ABB RobotStudio station: HackZurich_20170915-223747.rsstn

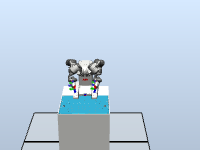
Station HackZurich (saved by RobotStudio 6.5.7530.2005)
Controller IRB_14000_0.5kg_0.5m_1, task T_ROB_L: task frame (RAPID world) sits at (0, 0, 832) mm in the station
Controller IRB_14000_0.5kg_0.5m_1, task T_ROB_R: task frame (RAPID world) sits at (0, 0, 832) mm in the station
Controller IRB_14000_0.5kg_0.5m_1
  mechanical unit ROB_R: IRB14000_0.5_0.5_R, 6 joints, base frame (0, 0, 0) mm
  mechanical unit ROB_R_7: IRB14000_0.5_0.5_R, 1 joints, base frame (0, 0, 0) mm
  mechanical unit ROB_L: IRB14000_0.5_0.5_L, 6 joints, base frame (0, 0, 0) mm
  mechanical unit ROB_L_7: IRB14000_0.5_0.5_L, 1 joints, base frame (0, 0, 0) mm
Layout (positions relative to the parent item):
  - SmartGripper_YuM_R [smart component] at (-9.58, -182.61, 1030.63) mm, rotated rx 179.34 ry -63.63 rz 15.45 deg
      signals: DI di_GripperClose, DI di_GripperOpen, GO SG_hand_ActualPosition, GO SG_hand_SysState, DO SG_hand_StatusCalibrated, GO SG_hand_SoftwareVersion, GO SG_hand_ActualSpeed, GI SG_hand_CmdGripper, GI SG_hand_MaxPosition, GI SG_hand_MinPosition
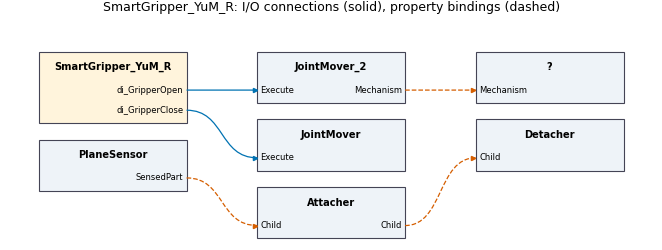
      connections:
        SmartGripper_YuM_R.di_GripperOpen -> JointMover_2.Execute
        SmartGripper_YuM_R.di_GripperClose -> JointMover.Execute
        PlaneSensor.SensedPart => Attacher.Child
        Attacher.Child => Detacher.Child
        JointMover_2.Mechanism => ?.Mechanism
    - PlaneSensor [smart component, from Components\PlaneSensor.rslib]
        properties: Origin=[-0.01 0 0.1]; Axis1=[0 0 0.03]; Axis2=[0.02 0 0]; SensedPart=DownFinger
      - _sensorPart_ [part]
    - Attacher [smart component, from Components\Attacher.rslib]
        properties: Parent=(none); Flange=0; Child=DownFinger; Mount=false; Offset=[0 0 0]; Orientation=[0 0 0]
    - Detacher [smart component, from Components\Detacher.rslib]
        properties: Child=DownFinger; KeepPosition=true
    - JointMover [smart component, from Components\JointMover.rslib]
        properties: Mechanism=YuMi_Hand_R; Relative=false; Duration=1; J1=0
    - JointMover_2 [smart component, from Components\JointMover.rslib]
        properties: Mechanism=YuMi_Hand_R; Relative=false; Duration=1; J1=0.025
    - YuMi_Hand_R [mechanism] at (0, 0, 0) mm; joint values [0] (rad or m)
        TCP Servo at (0, 0, 114.2) mm
        TCP VaccumOne at (56, 18.5, 37.5) mm, rotated rx 0 ry 90 rz 0 deg
        TCP Camera at (-7.3, 28.3, 35.1) mm, rotated rx 0 ry 90 rz 90 deg
        links: HandBase, DownFinger, UpFinger
  - SmartGripper_YuMi_L [smart component] at (-9.58, 182.61, 1030.63) mm, rotated rx -179.34 ry -63.63 rz -15.45 deg
      signals: DI di_GripperClose, DI di_GripperOpen, GO SG_hand_ActualPosition, GO SG_hand_SysState, DO SG_hand_StatusCalibrated, GO SG_hand_SoftwareVersion, GO SG_hand_ActualSpeed, GI SG_hand_CmdGripper, GI SG_hand_MaxPosition, GI SG_hand_MinPosition
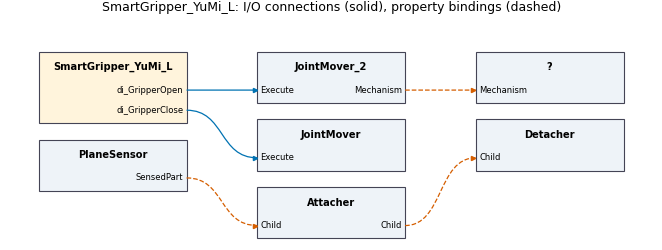
      connections:
        SmartGripper_YuMi_L.di_GripperOpen -> JointMover_2.Execute
        SmartGripper_YuMi_L.di_GripperClose -> JointMover.Execute
        PlaneSensor.SensedPart => Attacher.Child
        Attacher.Child => Detacher.Child
        JointMover_2.Mechanism => ?.Mechanism
    - PlaneSensor [smart component, from Components\PlaneSensor.rslib]
        properties: Origin=[-0.01 0 0.1]; Axis1=[0 0 0.03]; Axis2=[0.02 0 0]; SensedPart=DownFinger
      - _sensorPart_ [part]
    - Attacher [smart component, from Components\Attacher.rslib]
        properties: Parent=(none); Flange=0; Child=DownFinger; Mount=false; Offset=[0 0 0]; Orientation=[0 0 0]
    - Detacher [smart component, from Components\Detacher.rslib]
        properties: Child=DownFinger; KeepPosition=true
    - JointMover [smart component, from Components\JointMover.rslib]
        properties: Mechanism=YuMi_Hand_R; Relative=false; Duration=1; J1=0
    - JointMover_2 [smart component, from Components\JointMover.rslib]
        properties: Mechanism=YuMi_Hand_R; Relative=false; Duration=1; J1=0.025
    - YuMi_Hand_R [mechanism] at (0, 0, 0) mm; joint values [0] (rad or m)
        TCP Servo at (0, 0, 114.2) mm
        TCP VaccumOne at (56, 18.5, 37.5) mm, rotated rx 0 ry 90 rz 0 deg
        TCP Camera at (-7.3, 28.3, 35.1) mm, rotated rx 0 ry 90 rz 90 deg
        links: HandBase, DownFinger, UpFinger
  - IRB14000_0.5_0.5 [mechanism, from Robots\IRB14000_0.5_0.5__01.rslib] at (0, 0, 832) mm
  - IRB14000_0.5_0.5_R [mechanism, from Robots\IRB14000_0.5_0.5__01.rslib] at (0, 0, 832) mm; joint values [0, -2.2689, -2.3562, 0.5236, 0, 0.6981, 0] (rad or m)
  - IRB14000_0.5_0.5_L [mechanism, from Robots\IRB14000_0.5_0.5__01.rslib] at (0, 0, 832) mm; joint values [0, -2.2689, 2.3562, 0.5236, 0, 0.6981, 0] (rad or m)
  - 3HDA000058A6697 | YuMi-Tisch |   Lead Through mit Heberollen [graphiccomponentgroup] at (563, -309.12, 0) mm, rotated rx 0 ry 0 rz 94.33 deg
    - 3HDA000058A6699 | Rahmengestell |   YuMi:1 [graphiccomponentgroup]
      - 3HDA000058A4123 | ITEM Profil8 40x40 |  PROFIL 8 40X40 LEICHT, NATUR:1 [part] at (577.2, -60.29, 36) mm, rotated rx 0 ry -90 rz -3.99 deg
      - 3HDA000058A4123 | ITEM Profil8 40x40 |  PROFIL 8 40X40 LEICHT, NATUR:2 [part] at (577.2, -60.29, 796) mm, rotated rx 0 ry -90 rz -3.99 deg
      - 3HDA000057A1904 |Winkelsatz 8 |  WINKELSATZ 8 80X80 80x80:32 [part] at (621.28, -3.21, 736) mm, rotated rx 180 ry 0 rz 86.01 deg
      - 3HDA000057A1904 |Winkelsatz 8 |  WINKELSATZ 8 80X80 80x80:33 [part] at (716.12, 782.09, 736) mm, rotated rx 180 ry 0 rz -93.99 deg
      - 3HDA000057A1904 |Winkelsatz 8 |  WINKELSATZ 8 80X80 80x80:36 [part] at (-37.12, 42.68, 736) mm, rotated rx 180 ry 0 rz 86.01 deg
      - 3HDA000057A1904 |Winkelsatz 8 |  WINKELSATZ 8 80X80 80x80:37 [part] at (57.72, 827.99, 736) mm, rotated rx 180 ry 0 rz -93.99 deg
      - 3HDA000058A4120 | ITEM Profil 80x80 |  PROFIL 8X80X80 LEICHT leicht:1 [part] at (654.66, 475.62, 776) mm, rotated rx 0 ry -90 rz -3.99 deg
      - 3HDA000058A4119 | Hilfsprofil_Item_8_80x40_leicht |   L=615:1 [part] at (-17.17, 41.29, 776) mm, rotated rx 0 ry -90 rz -93.99 deg
      - 3HDA000058A4119 | Hilfsprofil_Item_8_80x40_leicht |   L=615:2 [part] at (696.17, 783.48, 776) mm, rotated rx 0 ry 90 rz -93.99 deg
      - 3HDA000058A4121 | ITEM Profil8 40x40 |  PROFIL 8 40X40 LEICHT, NATUR:3 [part] at (-17.17, 41.29, 36) mm, rotated rx -90 ry 0 rz -3.99 deg
      - 3HDA000058A4122 | ITEM Profil8 40x40 |  PROFIL 8 40X40 LEICHT, NATUR:1 [part] at (656.05, 495.58, 36) mm, rotated rx 0 ry -90 rz -3.99 deg
      - 3HDA000058A4121 | ITEM Profil8 40x40 |  PROFIL 8 40X40 LEICHT, NATUR:4 [part] at (641.23, -4.6, 36) mm, rotated rx -90 ry 0 rz -3.99 deg
      - 3HDA000058A6700 | ITEM Profil 80x80 |  PROFIL 8X80X80 LEICHT leicht:1 [part] at (0, 0, 0) mm, rotated rx 0 ry 0 rz -3.99 deg
      - Transport und Fußplatte 8 | 3HDA000001A5155 |  :1 [part] at (-37.12, 42.68, 0) mm, rotated rx 180 ry 0 rz -3.99 deg
      - 3HDA000058A6700 | ITEM Profil 80x80 |  PROFIL 8X80X80 LEICHT leicht:2 [part] at (618.5, -43.12, 0) mm, rotated rx 0 ry 0 rz -3.99 deg
      - Transport und Fußplatte 8 | 3HDA000001A5155 |  :2 [part] at (581.38, -0.43, 0) mm, rotated rx 180 ry 0 rz -3.99 deg
      - 3HDA000058A6700 | ITEM Profil 80x80 |  PROFIL 8X80X80 LEICHT leicht:3 [part] at (60.5, 867.89, 0) mm, rotated rx 0 ry 0 rz -3.99 deg
      - Transport und Fußplatte 8 | 3HDA000001A5155 |  :3 [part] at (23.38, 910.58, 0) mm, rotated rx 180 ry 0 rz -3.99 deg
      - 3HDA000058A6700 | ITEM Profil 80x80 |  PROFIL 8X80X80 LEICHT leicht:4 [part] at (679, 824.78, 0) mm, rotated rx 0 ry 0 rz -3.99 deg
      - Transport und Fußplatte 8 | 3HDA000001A5155 |  :4 [part] at (641.88, 867.46, 0) mm, rotated rx 180 ry 0 rz -3.99 deg
      - 3HDA000058A4123 | ITEM Profil8 40x40 |  PROFIL 8 40X40 LEICHT, NATUR:4 [part] at (101.8, 885.06, 36) mm, rotated rx 0 ry 90 rz -3.99 deg
      - Abdeckkappe 8 80x80 | 3HDA000000A3512 |  :1 [part] at (17.82, 830.77, 816) mm, rotated rx 0 ry 0 rz -3.99 deg
      - Abdeckkappe 8 80x80 | 3HDA000000A3512 |  :2 [part] at (636.32, 787.66, 816) mm, rotated rx 0 ry 0 rz -3.99 deg
      - 3HDA000058A4123 | ITEM Profil8 40x40 |  PROFIL 8 40X40 LEICHT, NATUR:5 [part] at (101.8, 885.06, 536) mm, rotated rx 0 ry 90 rz -3.99 deg
      - 3HDA000058A5960 | Heberolle |  HEBEROLLE D62 D62 - Hub 12mm:1 [part] at (0, 0, -16) mm, rotated rx 0 ry 0 rz 176.01 deg
      - 3HDA000058A5960 | Heberolle |  HEBEROLLE D62 D62 - Hub 12mm:2 [part] at (618.5, -43.12, -16) mm, rotated rx 0 ry 0 rz 176.01 deg
      - 3HDA000058A5960 | Heberolle |  HEBEROLLE D62 D62 - Hub 12mm:3 [part] at (60.5, 867.89, -16) mm, rotated rx 0 ry 0 rz -3.99 deg
      - 3HDA000058A5960 | Heberolle |  HEBEROLLE D62 D62 - Hub 12mm:4 [part] at (679, 824.78, -16) mm, rotated rx 0 ry 0 rz -3.99 deg
    - 3HDA000058A2017 | Arbeitsplatte |:1 [part] at (327.33, 237.81, 816) mm, rotated rx 0 ry 0 rz -3.99 deg
    - YuMi Tisch Verkleidung [part] at (350.71, 538.08, 10) mm, rotated rx 0 ry 0 rz -94.33 deg
    - Obere Abdeckung 1 [part] at (567.11, 879.93, 820) mm, rotated rx 0 ry 0 rz -94.33 deg
    - Obere Abdeckung 2 [part] at (18.68, 921.41, 820) mm, rotated rx 0 ry 0 rz -94.33 deg
Attachment: SmartGripper_YuM_R is attached to IRB14000_0.5_0.5_R / Link7
Attachment: SmartGripper_YuMi_L is attached to IRB14000_0.5_0.5_L / Link7
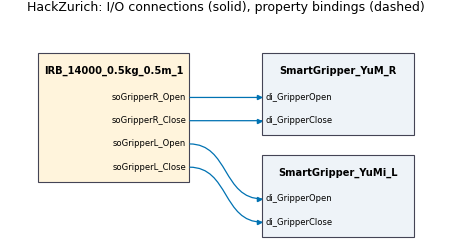
Station logic (signal -> signal, property => property):
  IRB_14000_0.5kg_0.5m_1.soGripperR_Open -> SmartGripper_YuM_R.di_GripperOpen
  IRB_14000_0.5kg_0.5m_1.soGripperR_Close -> SmartGripper_YuM_R.di_GripperClose
  IRB_14000_0.5kg_0.5m_1.soGripperL_Open -> SmartGripper_YuMi_L.di_GripperOpen
  IRB_14000_0.5kg_0.5m_1.soGripperL_Close -> SmartGripper_YuMi_L.di_GripperClose
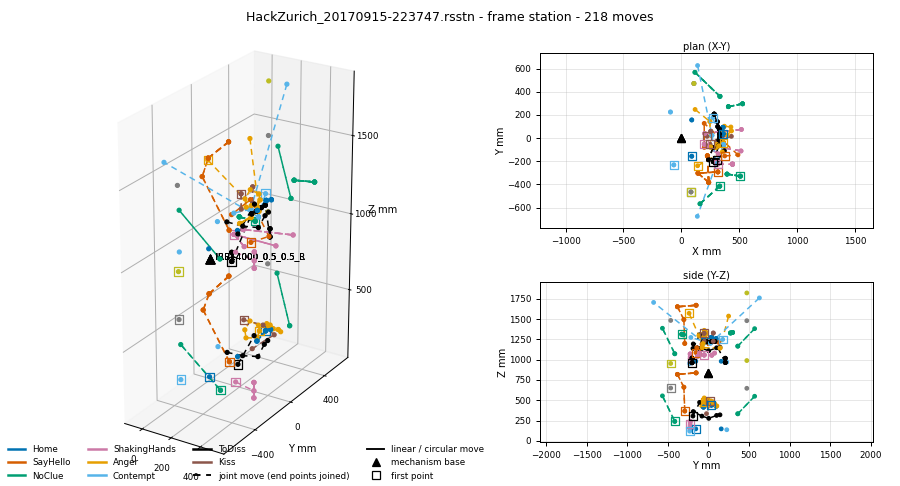
[picture p0: tool path of HackZurich_20170915-223747.rsstn in frame station, 218 of 222 moves have a stored position in this frame; points joined in program order, loops and branches not executed]
Targets, tools, work objects and paths stored in the station, written as RAPID:
! task T_ROB_R
MODULE GesturesRight
  CONST robtarget pKissR_10:=[[221.654761882,15.032417216,486.855961247],[0.69462356,-0.026998762,-0.017404571,0.718655868],[1,0,-2,4],[-163.076395011,9E+09,9E+09,9E+09,9E+09,9E+09]];
  CONST robtarget pKissR_20:=[[354.929073971,15.031772271,486.855510206],[0.677332175,0.151651856,0.155002452,0.702991521],[1,1,-2,4],[-128.711073694,9E+09,9E+09,9E+09,9E+09,9E+09]];
  CONST robtarget pKissR_30:=[[431.669236847,15.031318104,443.566889626],[0.639190619,0.273714512,0.272469802,0.665038289],[1,1,-2,4],[-128.711078258,9E+09,9E+09,9E+09,9E+09,9E+09]];
  CONST robtarget pKissR_40:=[[305.18930413,-24.552371649,335.517713502],[0.817106929,-0.136325958,0.414031132,0.377266114],[1,0,-2,4],[-146.11021025,9E+09,9E+09,9E+09,9E+09,9E+09]];
  CONST robtarget pAngerR_10:=[[363.531838424,-38.636637831,473.352200394],[0.300745531,-0.136482013,-0.04783233,-0.94267537],[1,0,0,4],[-130.403991592,9E+09,9E+09,9E+09,9E+09,9E+09]];
  CONST robtarget pAngerR_20:=[[350.75125662,-29.515051373,503.763471562],[0.257706669,0.015454476,-0.043694396,-0.965110995],[1,0,0,4],[-121.508331805,9E+09,9E+09,9E+09,9E+09,9E+09]];
  CONST robtarget pAngerR_30:=[[306.632986283,-52.601439571,528.928808016],[0.261410738,0.064341961,-0.04557113,-0.96200198],[1,0,0,4],[-122.099256333,9E+09,9E+09,9E+09,9E+09,9E+09]];
  CONST robtarget pAngerR_40:=[[288.800844629,-81.29752225,478.773158089],[0.216079199,-0.014900154,-0.132940712,-0.967168306],[1,0,0,4],[-129.63023687,9E+09,9E+09,9E+09,9E+09,9E+09]];
  CONST robtarget pAngerR_50:=[[297.418539835,-81.958124122,428.713986694],[0.109438137,-0.189120514,-0.255285462,-0.941852461],[1,0,0,4],[-136.020526211,9E+09,9E+09,9E+09,9E+09,9E+09]];
  CONST robtarget pAngerR_60:=[[354.350248531,-52.04234992,430.466884854],[0.177313873,-0.133250362,-0.160013373,-0.961873096],[1,0,0,4],[-129.960312977,9E+09,9E+09,9E+09,9E+09,9E+09]];
  CONST robtarget pContemptR_10:=[[-65.408295514,-231.499226874,119.303275828],[0.188476781,-0.180789855,-0.941418807,0.213359232],[1,0,-1,5],[-169.723005722,9E+09,9E+09,9E+09,9E+09,9E+09]];
  CONST robtarget pSayHelloR_10:=[[314.699715633,-292.148031152,367.159687256],[0.159532666,0.511489136,0.162496176,0.828566947],[1,0,0,5],[-122.185137209,9E+09,9E+09,9E+09,9E+09,9E+09]];
  CONST robtarget pSayHelloR_20:=[[143.244207362,-303.049195945,660.697114826],[0.6530857,-0.147210566,0.221457786,0.70905893],[1,0,0,5],[154.264930282,9E+09,9E+09,9E+09,9E+09,9E+09]];
  CONST robtarget pSayHelloR_30:=[[235.909258765,-382.383017558,818.803192241],[0.490338864,0.057638645,0.190726209,0.848450999],[1,0,0,5],[-161.185793796,9E+09,9E+09,9E+09,9E+09,9E+09]];
  CONST robtarget pSayHelloR_40:=[[223.935861995,-152.493872643,837.018526473],[0.280171534,-0.02496644,0.413534074,0.865950436],[1,0,0,5],[-151.318897483,9E+09,9E+09,9E+09,9E+09,9E+09]];
  CONST robtarget pShakingHandsR_10:=[[315.738569474,-225.378667241,206.19666017],[0.339537865,-0.658753284,0.219946518,-0.63433562],[0,0,1,4],[-108.735165241,9E+09,9E+09,9E+09,9E+09,9E+09]];
  CONST robtarget pShakingHandsR_40:=[[440.955889424,-225.380066174,182.362206426],[0.11092253,0.699479671,0.098185544,0.699130876],[1,1,-1,4],[-108.735179691,9E+09,9E+09,9E+09,9E+09,9E+09]];
  CONST robtarget pShakingHandsR_20:=[[440.955617046,-225.379654836,237.561937878],[0.110922498,0.699479548,0.098185209,0.699131051],[1,2,-1,4],[-108.735186134,9E+09,9E+09,9E+09,9E+09,9E+09]];
  CONST robtarget pShakingHandsR_30:=[[440.955691509,-225.379895287,135.696714265],[0.110922513,0.699479626,0.098185285,0.69913096],[1,1,-1,4],[-108.735178424,9E+09,9E+09,9E+09,9E+09,9E+09]];
  CONST robtarget pSuprisedR_10:=[[83.03148877,-465.085929834,650.386646622],[0.703838382,-0.01527703,0.013249227,-0.710072252],[1,0,-2,4],[115.639447021,9E+09,9E+09,9E+09,9E+09,9E+09]];
  CONST robtarget pHandsUpR_10:=[[83.03187344,-465.085940939,952.690090127],[0.703838421,-0.015277226,0.013249253,-0.710072208],[0,1,-2,4],[137.877026865,9E+09,9E+09,9E+09,9E+09,9E+09]];
  CONST robtarget pNoClueR_20:=[[331.005027183,-415.055262019,240.258080351],[0.395586627,0.754614135,0.446136315,0.273918084],[0,0,0,5],[-121.777862862,9E+09,9E+09,9E+09,9E+09,9E+09]];
  CONST robtarget pNoClueR_10:=[[160.547655799,-566.897146043,554.058433096],[0.765286197,0.45290272,-0.146899327,0.433170579],[1,0,0,5],[169.961367293,9E+09,9E+09,9E+09,9E+09,9E+09]];
  CONST robtarget pToDissR_10:=[[310.08261334,-191.393706007,305.466074161],[0.673664037,0.094173277,0.328608316,0.655228765],[1,0,-1,4],[-103.279379297,9E+09,9E+09,9E+09,9E+09,9E+09]];
  CONST robtarget pToDissR_20:=[[370.062778661,-109.65260016,473.851053749],[0.666629844,-0.160646787,-0.045141606,0.726470575],[1,0,-1,4],[-103.911686462,9E+09,9E+09,9E+09,9E+09,9E+09]];
  CONST robtarget pHomeR_10:=[[89.387946422,-156.622117956,147.913470217],[0.066010726,-0.842420918,-0.111214912,-0.523068661],[0,0,0,4],[-101.964427132,9E+09,9E+09,9E+09,9E+09,9E+09]];
  CONST robtarget pSayNoR_10:=[[359.801557873,36.119395579,442.32851368],[0.724497161,0.007725768,-0.00165855,-0.68923249],[1,0,0,4],[-143.857840595,9E+09,9E+09,9E+09,9E+09,9E+09]];
  CONST robtarget pSayNoR_20:=[[359.802142459,93.128614528,426.773071438],[0.708401181,-0.152065476,-0.153449882,-0.671935259],[1,0,0,4],[-143.857842721,9E+09,9E+09,9E+09,9E+09,9E+09]];
  CONST robtarget pSayNoR_30:=[[359.802673586,-61.261892837,415.421024536],[0.687551152,0.228536622,0.208835913,-0.656834824],[1,0,0,4],[-143.857842589,9E+09,9E+09,9E+09,9E+09,9E+09]];
  PROC Home()
    MoveJ pHomeR_10,v1000,fine,Servo\WObj:=wobj0;
  ENDPROC
  PROC SayHello()
    MoveJ pSayHelloR_10,v1000,z10,Servo\WObj:=wobj0;
    MoveJ pSayHelloR_20,v1000,z10,Servo\WObj:=wobj0;
    MoveJ pSayHelloR_30,v400,z10,Servo\WObj:=wobj0;
    MoveJ pSayHelloR_40,v400,z10,Servo\WObj:=wobj0;
    MoveJ pSayHelloR_30,v400,z10,Servo\WObj:=wobj0;
    MoveJ pSayHelloR_40,v400,z10,Servo\WObj:=wobj0;
    MoveJ pSayHelloR_40,v400,z10,Servo\WObj:=wobj0;
    MoveJ pSayHelloR_30,v400,z10,Servo\WObj:=wobj0;
    MoveJ pSayHelloR_20,v1000,z10,Servo\WObj:=wobj0;
    MoveJ pSayHelloR_10,v1000,z10,Servo\WObj:=wobj0;
    Home;
  ENDPROC
  PROC NoClue()
    MoveJ pNoClueR_20,v1000,z10,Servo\WObj:=wobj0;
    MoveJ pNoClueR_10,v1000,z10,Servo\WObj:=wobj0;
    WaitTime 2;
    MoveJ pNoClueR_20,v1000,z10,Servo\WObj:=wobj0;
    Home;
  ENDPROC
  PROC ShakingHands()
    MoveJ pShakingHandsR_10,v1000,z10,Servo\WObj:=wobj0;
    MoveJ pShakingHandsR_40,v1000,z10,Servo\WObj:=wobj0;
    WaitTime 1;
    MoveJ pShakingHandsR_20,v1000,z10,Servo\WObj:=wobj0;
    MoveJ pShakingHandsR_30,v1000,z10,Servo\WObj:=wobj0;
    MoveJ pShakingHandsR_20,v1000,z10,Servo\WObj:=wobj0;
    MoveJ pShakingHandsR_30,v1000,z10,Servo\WObj:=wobj0;
    MoveJ pShakingHandsR_20,v1000,z10,Servo\WObj:=wobj0;
    MoveJ pShakingHandsR_30,v1000,z10,Servo\WObj:=wobj0;
    MoveJ pShakingHandsR_40,v1000,z10,Servo\WObj:=wobj0;
    WaitTime 1;
    Home;
  ENDPROC
  PROC Anger()
    MoveJ pAngerR_10,v1000,z40,Servo\WObj:=wobj0;
    MoveJ pAngerR_20,v1000,z40,Servo\WObj:=wobj0;
    MoveJ pAngerR_30,v1000,z40,Servo\WObj:=wobj0;
    MoveJ pAngerR_40,v1000,z40,Servo\WObj:=wobj0;
    MoveJ pAngerR_50,v1000,z40,Servo\WObj:=wobj0;
    MoveJ pAngerR_60,v1000,z40,Servo\WObj:=wobj0;
    MoveJ pAngerR_10,v1000,z40,Servo\WObj:=wobj0;
    Home;
  ENDPROC
  PROC Contempt()
    MoveJ pContemptR_10,v1000,z10,Servo\WObj:=wobj0;
    WaitTime 2;
    Home;
  ENDPROC
  PROC ToDiss()
    MoveJ pToDissR_10,v500,z10,Servo\WObj:=wobj0;
    MoveJ pToDissR_20,v500,z10,Servo\WObj:=wobj0;
    WaitTime 1;
    Home;
  ENDPROC
  PROC Kiss()
    MoveJ pKissR_10,v1000,z10,Servo\WObj:=wobj0;
    MoveJ pKissR_20,v1000,z10,Servo\WObj:=wobj0;
    MoveJ pKissR_30,v1000,z10,Servo\WObj:=wobj0;
    MoveJ pKissR_40,v1000,z10,Servo\WObj:=wobj0;
    Home;
  ENDPROC
  PROC Suprised()
    MoveJ pSuprisedR_10,v5000,z10,Servo\WObj:=wobj0;
    WaitTime 2;
    Home;
  ENDPROC
  PROC HandsUp()
    MoveJ pHandsUpR_10,v1000,z10,Servo\WObj:=wobj0;
    WaitTime 2;
    Home;
  ENDPROC
  PROC SayNo()
    MoveJ pSayNoR_10,v1000,z10,Servo\WObj:=wobj0;
    MoveJ pSayNoR_20,v1000,z10,Servo\WObj:=wobj0;
    MoveJ pSayNoR_10,v1000,z10,Servo\WObj:=wobj0;
    MoveJ pSayNoR_30,v1000,z10,Servo\WObj:=wobj0;
    MoveJ pSayNoR_10,v1000,z10,Servo\WObj:=wobj0;
    MoveJ pSayNoR_20,v1000,z10,Servo\WObj:=wobj0;
    MoveJ pSayNoR_10,v1000,z10,Servo\WObj:=wobj0;
    MoveJ pSayNoR_30,v1000,z10,Servo\WObj:=wobj0;
    MoveJ pSayNoR_10,v1000,z10,Servo\WObj:=wobj0;
    MoveJ pSayNoR_20,v1000,z10,Servo\WObj:=wobj0;
    MoveJ pSayNoR_10,v1000,z10,Servo\WObj:=wobj0;
    MoveJ pSayNoR_30,v1000,z10,Servo\WObj:=wobj0;
    MoveJ pSayNoR_10,v1000,z10,Servo\WObj:=wobj0;
    Home;
  ENDPROC
ENDMODULE

! task T_ROB_R
MODULE user
  TASK PERS tooldata Servo:=[TRUE,[[0,0,114.2],[1,0,0,0]],[0.24,[8.2,12.5,48.1],[1,0,0,0],0.00022,0.00024,0.00009]];
ENDMODULE

! task T_ROB_L
MODULE GesturesLeft
  CONST robtarget pAngerL_10:=[[431.098301309,61.959159256,458.125646738],[0.188343319,-0.135994051,0.205422096,-0.950701938],[-1,0,1,4],[116.357977607,9E+09,9E+09,9E+09,9E+09,9E+09]];
  CONST robtarget pAngerL_20:=[[427.541303481,96.078854268,428.274281879],[0.242851724,-0.180947804,0.292829472,-0.906935407],[-1,0,1,4],[121.814803059,9E+09,9E+09,9E+09,9E+09,9E+09]];
  CONST robtarget pAngerL_30:=[[371.370802791,102.647922136,430.309317662],[0.250175091,-0.189729403,0.368594998,-0.874958802],[-1,0,1,4],[129.017692817,9E+09,9E+09,9E+09,9E+09,9E+09]];
  CONST robtarget pAngerL_40:=[[354.020430947,75.987991242,458.212372351],[0.211781199,-0.1200539,0.309854599,-0.919089719],[-1,0,1,4],[127.31237471,9E+09,9E+09,9E+09,9E+09,9E+09]];
  CONST robtarget pAngerL_50:=[[359.09325296,50.040718323,483.103930387],[0.132670971,-0.022575789,0.326351779,-0.935619187],[-1,0,1,4],[134.887718951,9E+09,9E+09,9E+09,9E+09,9E+09]];
  CONST robtarget pAngerL_60:=[[396.062972248,27.911166703,492.703033028],[0.114272503,-0.022558134,0.275782172,-0.954136845],[-1,0,1,4],[129.639362388,9E+09,9E+09,9E+09,9E+09,9E+09]];
  CONST robtarget pContemptL_10:=[[-94.491553607,225.077568886,137.327093089],[0.306193092,0.231227469,-0.892125882,-0.238518467],[-1,0,1,5],[170.068678796,9E+09,9E+09,9E+09,9E+09,9E+09]];
  CONST robtarget pSuprisedL_10:=[[108.153191894,471.411528047,647.230762026],[0.699371757,0.003098078,0.006552088,-0.714721357],[-1,0,0,4],[-132.382826108,9E+09,9E+09,9E+09,9E+09,9E+09]];
  CONST robtarget pHandsUpL_10:=[[108.153567372,471.411547841,988.720364525],[0.699371728,0.003098049,0.006552252,-0.714721384],[0,-1,0,4],[-132.382818416,9E+09,9E+09,9E+09,9E+09,9E+09]];
  CONST robtarget pNoClueL_20:=[[332.599072052,360.424339744,333.84998915],[0.323491568,-0.733582932,-0.040436016,-0.596300441],[-1,0,0,5],[100.391786771,9E+09,9E+09,9E+09,9E+09,9E+09]];
  CONST robtarget pNoClueL_10:=[[116.844170561,567.745373907,549.176802943],[0.612414859,-0.27944775,-0.40047322,-0.621673705],[-1,0,0,5],[170.97345488,9E+09,9E+09,9E+09,9E+09,9E+09]];
  CONST robtarget pToDissL_10:=[[311.262788205,141.365155063,320.620976131],[0.30127594,0.413850338,-0.12183377,0.850363004],[-1,0,0,4],[109.137922493,9E+09,9E+09,9E+09,9E+09,9E+09]];
  CONST robtarget pToDissL_20:=[[313.163869898,99.550091581,313.678214603],[0.405584331,0.369718383,-0.180052484,0.816327612],[-1,0,0,4],[120.550323233,9E+09,9E+09,9E+09,9E+09,9E+09]];
  CONST robtarget pToDissL_30:=[[327.793203037,3.134311337,277.462215839],[0.525517576,0.35593926,-0.443885036,0.632538216],[-1,0,0,4],[161.707001678,9E+09,9E+09,9E+09,9E+09,9E+09]];
  CONST robtarget pToDissL_40:=[[274.023321791,-80.991562457,305.086937965],[0.647848865,0.227051384,-0.451204352,0.570222895],[-1,0,0,4],[171.12747593,9E+09,9E+09,9E+09,9E+09,9E+09]];
  CONST robtarget pToDissL_50:=[[233.086731165,-187.421735572,361.300083015],[0.647848463,0.227050931,-0.451204503,0.570223413],[-1,1,-1,4],[154.498524311,9E+09,9E+09,9E+09,9E+09,9E+09]];
  CONST robtarget pHomeL_10:=[[89.387946423,156.622117957,147.913470217],[0.066010726,0.842420918,-0.111214912,0.523068661],[0,0,0,4],[101.964427132,9E+09,9E+09,9E+09,9E+09,9E+09]];
  PROC Suprised()
    MoveJ pSuprisedL_10,v5000,z10,Servo\WObj:=wobj0;
    WaitTime 2;
    Home;
  ENDPROC
  PROC Contempt()
    MoveJ pContemptL_10,v1000,z10,Servo\WObj:=wobj0;
    WaitTime 2;
    Home;
  ENDPROC
  PROC Home()
    MoveJ pHomeL_10,v1000,fine,Servo\WObj:=wobj0;
  ENDPROC
  PROC NoClue()
    MoveJ pNoClueL_20,v1000,z10,Servo\WObj:=wobj0;
    MoveJ pNoClueL_10,v1000,z10,Servo\WObj:=wobj0;
    WaitTime 2;
    MoveJ pNoClueL_20,v1000,z10,Servo\WObj:=wobj0;
    Home;
  ENDPROC
  PROC ToDiss()
    MoveJ pToDissL_10,v1000,z10,Servo\WObj:=wobj0;
    MoveJ pToDissL_20,v1000,z10,Servo\WObj:=wobj0;
    MoveJ pToDissL_30,v1000,z10,Servo\WObj:=wobj0;
    MoveJ pToDissL_40,v1000,z10,Servo\WObj:=wobj0;
    MoveJ pToDissL_50,v1000,fine,Servo\WObj:=wobj0;
    WaitTime 1;
    Home;
  ENDPROC
  PROC Anger()
    MoveJ pAngerL_10,v1000,z40,Servo\WObj:=wobj0;
    MoveJ pAngerL_20,v1000,z40,Servo\WObj:=wobj0;
    MoveJ pAngerL_30,v1000,z40,Servo\WObj:=wobj0;
    MoveJ pAngerL_40,v1000,z40,Servo\WObj:=wobj0;
    MoveJ pAngerL_50,v1000,z40,Servo\WObj:=wobj0;
    MoveJ pAngerL_60,v1000,z40,Servo\WObj:=wobj0;
    MoveJ pAngerL_10,v1000,z40,Servo\WObj:=wobj0;
    Home;
  ENDPROC
  PROC HandsUp()
    MoveJ pHandsUpL_10,v1000,z10,Servo\WObj:=wobj0;
    WaitTime 2;
    Home;
  ENDPROC
ENDMODULE

! task T_ROB_L
MODULE user
  TASK PERS tooldata Servo:=[TRUE,[[0,0,114.2],[1,0,0,0]],[0.24,[8.2,12.5,48.1],[1,0,0,0],0.00022,0.00024,0.00009]];
ENDMODULE

! task T_ROB_R
MODULE Gestures
  CONST robtarget pHomeR_10:=[[89.387946422,-156.622117956,147.913470217],[0.066010726,-0.842420918,-0.111214912,-0.523068661],[0,0,0,4],[-101.964427132,9E+09,9E+09,9E+09,9E+09,9E+09]];
  CONST robtarget pSayHelloR_10:=[[314.699715633,-292.148031152,367.159687256],[0.159532666,0.511489136,0.162496176,0.828566947],[1,0,0,5],[-122.185137209,9E+09,9E+09,9E+09,9E+09,9E+09]];
  CONST robtarget pSayHelloR_20:=[[143.244207362,-303.049195945,660.697114826],[0.6530857,-0.147210566,0.221457786,0.70905893],[1,0,0,5],[154.264930282,9E+09,9E+09,9E+09,9E+09,9E+09]];
  CONST robtarget pSayHelloR_30:=[[235.909258765,-382.383017558,818.803192241],[0.490338864,0.057638645,0.190726209,0.848450999],[1,0,0,5],[-161.185793796,9E+09,9E+09,9E+09,9E+09,9E+09]];
  CONST robtarget pSayHelloR_40:=[[223.935861995,-152.493872643,837.018526473],[0.280171534,-0.02496644,0.413534074,0.865950436],[1,0,0,5],[-151.318897483,9E+09,9E+09,9E+09,9E+09,9E+09]];
  VAR syncident syncCommandStart;
  CONST robtarget pNoClueR_20:=[[331.005027183,-415.055262019,240.258080351],[0.395586627,0.754614135,0.446136315,0.273918084],[0,0,0,5],[-121.777862862,9E+09,9E+09,9E+09,9E+09,9E+09]];
  CONST robtarget pNoClueR_10:=[[160.547655799,-566.897146043,554.058433096],[0.765286197,0.45290272,-0.146899327,0.433170579],[1,0,0,5],[169.961367293,9E+09,9E+09,9E+09,9E+09,9E+09]];
  CONST robtarget pShakingHandsR_10:=[[315.738569474,-225.378667241,206.19666017],[0.339537865,-0.658753284,0.219946518,-0.63433562],[0,0,1,4],[-108.735165241,9E+09,9E+09,9E+09,9E+09,9E+09]];
  CONST robtarget pShakingHandsR_40:=[[440.955889424,-225.380066174,182.362206426],[0.11092253,0.699479671,0.098185544,0.699130876],[1,1,-1,4],[-108.735179691,9E+09,9E+09,9E+09,9E+09,9E+09]];
  CONST robtarget pShakingHandsR_20:=[[440.955617046,-225.379654836,237.561937878],[0.110922498,0.699479548,0.098185209,0.699131051],[1,2,-1,4],[-108.735186134,9E+09,9E+09,9E+09,9E+09,9E+09]];
  CONST robtarget pShakingHandsR_30:=[[440.955691509,-225.379895287,135.696714265],[0.110922513,0.699479626,0.098185285,0.69913096],[1,1,-1,4],[-108.735178424,9E+09,9E+09,9E+09,9E+09,9E+09]];
  CONST robtarget pAngerR_10:=[[363.531838424,-38.636637831,473.352200394],[0.300745531,-0.136482013,-0.04783233,-0.94267537],[1,0,0,4],[-130.403991592,9E+09,9E+09,9E+09,9E+09,9E+09]];
  CONST robtarget pAngerR_20:=[[350.75125662,-29.515051373,503.763471562],[0.257706669,0.015454476,-0.043694396,-0.965110995],[1,0,0,4],[-121.508331805,9E+09,9E+09,9E+09,9E+09,9E+09]];
  CONST robtarget pAngerR_30:=[[306.632986283,-52.601439571,528.928808016],[0.261410738,0.064341961,-0.04557113,-0.96200198],[1,0,0,4],[-122.099256333,9E+09,9E+09,9E+09,9E+09,9E+09]];
  CONST robtarget pAngerR_40:=[[288.800844629,-81.29752225,478.773158089],[0.216079199,-0.014900154,-0.132940712,-0.967168306],[1,0,0,4],[-129.63023687,9E+09,9E+09,9E+09,9E+09,9E+09]];
  CONST robtarget pAngerR_50:=[[297.418539835,-81.958124122,428.713986694],[0.109438137,-0.189120514,-0.255285462,-0.941852461],[1,0,0,4],[-136.020526211,9E+09,9E+09,9E+09,9E+09,9E+09]];
  CONST robtarget pAngerR_60:=[[354.350248531,-52.04234992,430.466884854],[0.177313873,-0.133250362,-0.160013373,-0.961873096],[1,0,0,4],[-129.960312977,9E+09,9E+09,9E+09,9E+09,9E+09]];
  CONST robtarget pContemptR_10:=[[-65.408295514,-231.499226874,119.303275828],[0.188476781,-0.180789855,-0.941418807,0.213359232],[1,0,-1,5],[-169.723005722,9E+09,9E+09,9E+09,9E+09,9E+09]];
  CONST robtarget pToDissR_10:=[[310.08261334,-191.393706007,305.466074161],[0.673664037,0.094173277,0.328608316,0.655228765],[1,0,-1,4],[-103.279379297,9E+09,9E+09,9E+09,9E+09,9E+09]];
  CONST robtarget pToDissR_20:=[[370.062778661,-109.65260016,473.851053749],[0.666629844,-0.160646787,-0.045141606,0.726470575],[1,0,-1,4],[-103.911686462,9E+09,9E+09,9E+09,9E+09,9E+09]];
  VAR syncident syncToDiss;
  CONST robtarget pKissR_10:=[[221.654761882,15.032417216,486.855961247],[0.69462356,-0.026998762,-0.017404571,0.718655868],[1,0,-2,4],[-163.076395011,9E+09,9E+09,9E+09,9E+09,9E+09]];
  CONST robtarget pKissR_20:=[[354.929073971,15.031772271,486.855510206],[0.677332175,0.151651856,0.155002452,0.702991521],[1,1,-2,4],[-128.711073694,9E+09,9E+09,9E+09,9E+09,9E+09]];
  CONST robtarget pKissR_30:=[[431.669236847,15.031318104,443.566889626],[0.639190619,0.273714512,0.272469802,0.665038289],[1,1,-2,4],[-128.711078258,9E+09,9E+09,9E+09,9E+09,9E+09]];
  CONST robtarget pKissR_40:=[[305.18930413,-24.552371649,335.517713502],[0.817106929,-0.136325958,0.414031132,0.377266114],[1,0,-2,4],[-146.11021025,9E+09,9E+09,9E+09,9E+09,9E+09]];
  CONST robtarget pSuprisedR_10:=[[83.03148877,-465.085929834,650.386646622],[0.703838382,-0.01527703,0.013249227,-0.710072252],[1,0,-2,4],[115.639447021,9E+09,9E+09,9E+09,9E+09,9E+09]];
  CONST robtarget pHandsUpR_10:=[[83.03187344,-465.085940939,952.690090127],[0.703838421,-0.015277226,0.013249253,-0.710072208],[0,1,-2,4],[137.877026865,9E+09,9E+09,9E+09,9E+09,9E+09]];
  CONST robtarget pSayNoR_10:=[[359.801557873,36.119395579,442.32851368],[0.724497161,0.007725768,-0.00165855,-0.68923249],[1,0,0,4],[-143.857840595,9E+09,9E+09,9E+09,9E+09,9E+09]];
  CONST robtarget pSayNoR_20:=[[359.802142459,93.128614528,426.773071438],[0.708401181,-0.152065476,-0.153449882,-0.671935259],[1,0,0,4],[-143.857842721,9E+09,9E+09,9E+09,9E+09,9E+09]];
  CONST robtarget pSayNoR_30:=[[359.802673586,-61.261892837,415.421024536],[0.687551152,0.228536622,0.208835913,-0.656834824],[1,0,0,4],[-143.857842589,9E+09,9E+09,9E+09,9E+09,9E+09]];
  CONST robtarget pIKillYou10:=[[374.16,-154.35,254.16],[0.161557,0.694401,0.0894066,0.695495],[1,1,-1,4],[-117.393,9E+09,9E+09,9E+09,9E+09,9E+09]];
  CONST robtarget pIKillYou20:=[[488.56,-144.83,314.81],[0.000395089,-0.719169,-0.00618865,-0.694808],[1,2,-2,4],[-101.713,9E+09,9E+09,9E+09,9E+09,9E+09]];
  CONST robtarget pIKillYou30:=[[196.92,127.33,379.19],[0.180402,0.188619,-0.483007,-0.835812],[1,1,-2,5],[-129.125,9E+09,9E+09,9E+09,9E+09,9E+09]];
  CONST robtarget pIKillYou40:=[[197.77,-80.86,359.78],[0.278102,0.15155,-0.466809,-0.8257],[1,2,-2,5],[-126.747,9E+09,9E+09,9E+09,9E+09,9E+09]];
  CONST robtarget pGiveMeAHug10:=[[509.34,-328.38,480.34],[0.155829,0.0974494,0.882897,0.432104],[0,0,0,4],[155.094,9E+09,9E+09,9E+09,9E+09,9E+09]];
  VAR syncident syncGiveMeAHug;
  CONST robtarget pGiveMeAHug20:=[[393.96,-310.78,474.19],[0.193899,0.0762726,-0.873009,-0.440955],[0,0,0,4],[156.47,9E+09,9E+09,9E+09,9E+09,9E+09]];
  VAR syncident syncGiveMeAHug1;
  VAR syncident syncGoAway;
  CONST robtarget pGoAway10:=[[197.61,-52.8,224.96],[0.499064,-0.586453,-0.400827,-0.496333],[0,-1,1,4],[-116.88,9E+09,9E+09,9E+09,9E+09,9E+09]];
  CONST robtarget pGoAway20:=[[514.65,-111.17,249.33],[0.259577,-0.6352,-0.212178,-0.695788],[1,-1,1,4],[-120.721,9E+09,9E+09,9E+09,9E+09,9E+09]];
  VAR syncident syncGoAway1;
  CONST robtarget pGoAway30:=[[317.99,-135.96,207.81],[0.221309,-0.723273,-0.258737,-0.600794],[0,-1,1,4],[-117.948,9E+09,9E+09,9E+09,9E+09,9E+09]];
  VAR syncident syncGoAway2;
  CONST robtarget pPowerfull10:=[[140.08,-238.76,738.33],[0.454908,-0.375862,0.550802,0.590257],[1,0,0,4],[173.484,9E+09,9E+09,9E+09,9E+09,9E+09]];
  CONST robtarget pPowerfull20:=[[353.35,-118.73,464.57],[0.235961,-0.363756,-0.103651,0.895131],[1,0,0,4],[-87.9474,9E+09,9E+09,9E+09,9E+09,9E+09]];
  VAR syncident syncPowerfull;
  CONST robtarget pHappy10:=[[270.72,174.42,416.02],[0.424616,-0.16407,-0.415377,-0.787556],[1,0,0,4],[-156.077,9E+09,9E+09,9E+09,9E+09,9E+09]];
  VAR syncident syncHappy;
  CONST robtarget pHappy20:=[[362.98,-54.19,373.08],[0.14727,-0.120428,-0.717561,-0.670012],[0,0,0,4],[174.558,9E+09,9E+09,9E+09,9E+09,9E+09]];
  VAR syncident syncHappy1;
  VAR syncident syncHappy2;
  CONST robtarget pHappy30:=[[137.55,-675.5,871.93],[0.696123,0.382261,0.348089,-0.49812],[0,0,0,6],[50.4932,9E+09,9E+09,9E+09,9E+09,9E+09]];
  VAR syncident syncHappy3;
  CONST robtarget pExcited10:=[[275.33,-202.51,129.63],[0.0269036,-0.723872,-0.129753,-0.677089],[0,0,0,4],[-106.838,9E+09,9E+09,9E+09,9E+09,9E+09]];
  VAR syncident syncExcited;
  CONST robtarget pExcited20:=[[275.24,-202.41,186.57],[0.0270641,-0.723988,-0.12976,-0.676958],[0,0,0,4],[-106.853,9E+09,9E+09,9E+09,9E+09,9E+09]];
  VAR syncident syncExcited1;
  CONST robtarget pExcited30:=[[323.93,-65.42,387.99],[0.517684,-0.471011,0.505859,0.50424],[1,-1,-1,4],[-106.11,9E+09,9E+09,9E+09,9E+09,9E+09]];
  VAR syncident syncExcited2;
  CONST robtarget pExcited40:=[[325.27,-16.87,386.93],[0.51709,-0.469045,0.507547,0.504986],[1,-1,0,4],[-106.069,9E+09,9E+09,9E+09,9E+09,9E+09]];
  VAR syncident syncExcited3;
  CONST robtarget pScared10:=[[245.99,-54.68,490.9],[0.711197,-0.0374195,-0.0510866,0.700135],[1,0,-1,4],[-114.575,9E+09,9E+09,9E+09,9E+09,9E+09]];
  VAR syncident syncScared;
  CONST robtarget pScared20:=[[246.96,-54.06,395.22],[0.711164,-0.0365424,-0.0478151,0.700446],[1,0,-1,4],[-114.624,9E+09,9E+09,9E+09,9E+09,9E+09]];
  VAR syncident syncScared1;
  PROC Home()
    MoveJ pHomeR_10,v1000,fine,Servo\WObj:=wobj0;
  ENDPROC
  PROC SayHello()
    MoveJ pSayHelloR_10,v1000,z10,Servo\WObj:=wobj0;
    MoveJ pSayHelloR_20,v1000,z10,Servo\WObj:=wobj0;
    MoveJ pSayHelloR_30,v400,z10,Servo\WObj:=wobj0;
    MoveJ pSayHelloR_40,v400,z10,Servo\WObj:=wobj0;
    MoveJ pSayHelloR_30,v400,z10,Servo\WObj:=wobj0;
    MoveJ pSayHelloR_40,v400,z10,Servo\WObj:=wobj0;
    MoveJ pSayHelloR_40,v400,z10,Servo\WObj:=wobj0;
    MoveJ pSayHelloR_30,v400,z10,Servo\WObj:=wobj0;
    MoveJ pSayHelloR_20,v1000,z10,Servo\WObj:=wobj0;
    MoveJ pSayHelloR_10,v1000,z10,Servo\WObj:=wobj0;
    Home;
  ENDPROC
  PROC NoClue()
    WaitSyncTask syncCommandStart,task_list\TimeOut:=5;
    MoveJ pNoClueR_20,v1000,z10,Servo\WObj:=wobj0;
    MoveJ pNoClueR_10,v1000,fine,Servo\WObj:=wobj0;
    WaitTime 2;
    MoveJ pNoClueR_20,v1000,z10,Servo\WObj:=wobj0;
    Home;
  ENDPROC
  PROC ShakingHands()
    MoveJ pShakingHandsR_10,v1000,z10,Servo\WObj:=wobj0;
    MoveJ pShakingHandsR_40,v1000,z10,Servo\WObj:=wobj0;
    WaitTime 1;
    MoveJ pShakingHandsR_20,v1000,z10,Servo\WObj:=wobj0;
    MoveJ pShakingHandsR_30,v1000,z10,Servo\WObj:=wobj0;
    MoveJ pShakingHandsR_20,v1000,z10,Servo\WObj:=wobj0;
    MoveJ pShakingHandsR_30,v1000,z10,Servo\WObj:=wobj0;
    MoveJ pShakingHandsR_20,v1000,z10,Servo\WObj:=wobj0;
    MoveJ pShakingHandsR_30,v1000,z10,Servo\WObj:=wobj0;
    MoveJ pShakingHandsR_40,v1000,z10,Servo\WObj:=wobj0;
    WaitTime 1;
    Home;
  ENDPROC
  PROC Anger()
    WaitSyncTask syncCommandStart,task_list\TimeOut:=5;
    MoveJ pAngerR_10,v1000,z40,Servo\WObj:=wobj0;
    MoveJ pAngerR_20,v1000,z40,Servo\WObj:=wobj0;
    MoveJ pAngerR_30,v1000,z40,Servo\WObj:=wobj0;
    MoveJ pAngerR_40,v1000,z40,Servo\WObj:=wobj0;
    MoveJ pAngerR_50,v1000,z40,Servo\WObj:=wobj0;
    MoveJ pAngerR_60,v1000,z40,Servo\WObj:=wobj0;
    MoveJ pAngerR_10,v1000,z40,Servo\WObj:=wobj0;
    Home;
  ENDPROC
  PROC Contempt()
    WaitSyncTask syncCommandStart,task_list\TimeOut:=5;
    MoveJ pContemptR_10,v1000,fine,Servo\WObj:=wobj0;
    WaitTime 2;
    Home;
  ENDPROC
  PROC ToDiss()
    WaitSyncTask syncCommandStart,task_list\TimeOut:=5;
    MoveJ pToDissR_10,v500,z10,Servo\WObj:=wobj0;
    MoveJ pToDissR_20,v500,fine,Servo\WObj:=wobj0;
    WaitSyncTask syncToDiss,task_list;
    WaitTime 1;
    Home;
  ENDPROC
  PROC Suprised()
    WaitSyncTask syncCommandStart,task_list\TimeOut:=5;
    MoveJ pSuprisedR_10,v5000,fine,Servo\WObj:=wobj0;
    WaitTime 2;
    Home;
  ENDPROC
  PROC SayNo()
    MoveJ pSayNoR_10,v1000,z10,Servo\WObj:=wobj0;
    MoveJ pSayNoR_20,v1000,z10,Servo\WObj:=wobj0;
    MoveJ pSayNoR_10,v1000,z10,Servo\WObj:=wobj0;
    MoveJ pSayNoR_30,v1000,z10,Servo\WObj:=wobj0;
    MoveJ pSayNoR_10,v1000,z10,Servo\WObj:=wobj0;
    MoveJ pSayNoR_20,v1000,z10,Servo\WObj:=wobj0;
    MoveJ pSayNoR_10,v1000,z10,Servo\WObj:=wobj0;
    MoveJ pSayNoR_30,v1000,z10,Servo\WObj:=wobj0;
    MoveJ pSayNoR_10,v1000,z10,Servo\WObj:=wobj0;
    MoveJ pSayNoR_20,v1000,z10,Servo\WObj:=wobj0;
    MoveJ pSayNoR_10,v1000,z10,Servo\WObj:=wobj0;
    MoveJ pSayNoR_30,v1000,z10,Servo\WObj:=wobj0;
    MoveJ pSayNoR_10,v1000,z10,Servo\WObj:=wobj0;
    Home;
  ENDPROC
  PROC IKillYou()
    MoveJ pIKillYou10,v300,z10,Servo;
    MoveJ pIKillYou20,v1000,fine,Servo;
    WaitTime 2;
    MoveJ pIKillYou30,v1000,z10,Servo;
    MoveL pIKillYou40,v100,fine,Servo;
    WaitTime 2;
    Home;
  ENDPROC
  PROC GiveMeAHug()
    MoveJ pGiveMeAHug10,v1000,fine,Servo;
    WaitSyncTask syncGiveMeAHug,task_list;
    WaitTime 2;
    MoveJ pGiveMeAHug20,v1000,fine,Servo;
    MoveJ pGiveMeAHug10,v1000,fine,Servo;
    MoveJ pGiveMeAHug20,v1000,fine,Servo;
    MoveJ pGiveMeAHug10,v1000,fine,Servo;
    MoveJ pGiveMeAHug20,v1000,fine,Servo;
    MoveJ pGiveMeAHug10,v1000,fine,Servo;
    MoveJ pGiveMeAHug20,v1000,fine,Servo;
    WaitSyncTask syncGiveMeAHug1,task_list;
    WaitTime 2;
    Home;
  ENDPROC
  PROC GoAway()
    WaitSyncTask syncCommandStart,task_list\TimeOut:=5;
    SyncMoveOn syncGoAway,task_list;
    MoveJ pGoAway10\ID:=10,v1000,fine,Servo;
    MoveJ pGoAway20\ID:=20,v1000,fine,Servo;
    MoveJ pGoAway10\ID:=30,v1000,fine,Servo;
    MoveJ pGoAway20\ID:=40,v1000,fine,Servo;
    MoveJ pGoAway10\ID:=50,v1000,fine,Servo;
    SyncMoveOff syncGoAway1;
    WaitTime 2;
    MoveJ pGoAway30,v1000,fine,Servo;
    MoveJ pGoAway10,v1000,fine,Servo;
    MoveJ pGoAway30,v1000,fine,Servo;
    MoveJ pGoAway10,v1000,fine,Servo;
    WaitTime 2;
    WaitSyncTask syncGoAway2,task_list;
    Home;
  ENDPROC
  PROC Powerful()
    WaitSyncTask syncCommandStart,task_list\TimeOut:=5;
    MoveJ pPowerfull10,v1000,fine,Servo;
    WaitTime 2;
    MoveJ pPowerfull20,v1000,fine,Servo;
    WaitSyncTask syncPowerfull,task_list;
    Home;
  ENDPROC
  PROC Happy()
    WaitSyncTask syncCommandStart,task_list\TimeOut:=5;
    MoveJ pHappy10,v1000,fine,Servo;
    WaitTime 1;
    WaitSyncTask syncHappy,task_list;
    MoveJ pHappy20,v1000,fine,Servo;
    SyncMoveOn syncHappy1,task_list;
    MoveC Offs(pHappy20,-nCircleDiameter/2,0,-nCircleDiameter/2),Offs(pHappy20,-nCircleDiameter,0,0)\ID:=10,v1000,z5,Servo;
    MoveC Offs(pHappy20,-nCircleDiameter/2,0,nCircleDiameter/2),pHappy20\ID:=20,v1000,z5,Servo;
    MoveC Offs(pHappy20,-nCircleDiameter/2,0,-nCircleDiameter/2),Offs(pHappy20,-nCircleDiameter,0,0)\ID:=30,v1000,z5,Servo;
    MoveC Offs(pHappy20,-nCircleDiameter/2,0,nCircleDiameter/2),pHappy20\ID:=40,v1000,z5,Servo;
    SyncMoveOff syncHappy2;
    MoveJ pHappy30,v1000,fine,Servo;
    WaitTime 2;
    WaitSyncTask syncHappy3,task_list;
    Home;
  ENDPROC
  PROC Excited()
    WaitSyncTask syncCommandStart,task_list\TimeOut:=5;
    MoveJ pExcited10,v1000,fine,Servo;
    SyncMoveOn syncExcited,task_list;
    MoveJ pExcited20\ID:=10,v1000,z5,Servo;
    MoveJ pExcited10\ID:=20,v1000,z5,Servo;
    MoveJ pExcited20\ID:=30,v1000,z5,Servo;
    MoveJ pExcited10\ID:=40,v1000,z5,Servo;
    MoveJ pExcited20\ID:=50,v1000,z5,Servo;
    MoveJ pExcited10\ID:=60,v1000,fine,Servo;
    SyncMoveOff syncExcited1;
    WaitTime 1;
    MoveJ pExcited30,v1000,fine,Servo;
    WaitTime 0.5;
    SyncMoveOn syncExcited2,task_list;
    MoveJ pExcited40\ID:=10,v1000,z5,Servo;
    MoveJ pExcited30\ID:=20,v1000,z5,Servo;
    MoveJ pExcited40\ID:=30,v1000,z5,Servo;
    MoveJ pExcited30\ID:=40,v1000,z5,Servo;
    MoveJ pExcited40\ID:=50,v1000,z5,Servo;
    MoveJ pExcited30\ID:=60,v1000,fine,Servo;
    SyncMoveOff syncExcited3;
    WaitTime 2;
    Home;
  ENDPROC
  PROC Scared()
    WaitSyncTask syncCommandStart,task_list\TimeOut:=5;
    MoveJ pScared10,v1000,fine,Servo;
    WaitTime 2;
    SyncMoveOn syncScared,task_list;
    MoveJ pScared20\ID:=10,v100,fine,Servo;
    MoveJ pScared10\ID:=20,v1000,fine,Servo;
    SyncMoveOff syncScared1;
    WaitTime 2;
    Home;
  ENDPROC
ENDMODULE

! task T_ROB_R
MODULE Gripper_R
  PERS tooldata Servo:=[TRUE,[[0,0,114.2],[1,0,0,0]],[0.24,[8.2,12.5,48.1],[1,0,0,0],0.00022,0.00024,0.00009]];
ENDMODULE

! task T_ROB_R
MODULE MainModule
  PERS tasks task_list{2}:=[["T_ROB_R"], ["T_ROB_L"]];
ENDMODULE

! task T_ROB_L
MODULE Gestures
  CONST robtarget pHomeL_10:=[[89.387946423,156.622117957,147.913470217],[0.066010726,0.842420918,-0.111214912,0.523068661],[0,0,0,4],[101.964427132,9E+09,9E+09,9E+09,9E+09,9E+09]];
  VAR syncident syncCommandStart;
  CONST robtarget pAngerL_10:=[[431.098301309,61.959159256,458.125646738],[0.188343319,-0.135994051,0.205422096,-0.950701938],[-1,0,1,4],[116.357977607,9E+09,9E+09,9E+09,9E+09,9E+09]];
  CONST robtarget pAngerL_20:=[[427.541303481,96.078854268,428.274281879],[0.242851724,-0.180947804,0.292829472,-0.906935407],[-1,0,1,4],[121.814803059,9E+09,9E+09,9E+09,9E+09,9E+09]];
  CONST robtarget pAngerL_30:=[[371.370802791,102.647922136,430.309317662],[0.250175091,-0.189729403,0.368594998,-0.874958802],[-1,0,1,4],[129.017692817,9E+09,9E+09,9E+09,9E+09,9E+09]];
  CONST robtarget pAngerL_40:=[[354.020430947,75.987991242,458.212372351],[0.211781199,-0.1200539,0.309854599,-0.919089719],[-1,0,1,4],[127.31237471,9E+09,9E+09,9E+09,9E+09,9E+09]];
  CONST robtarget pAngerL_50:=[[359.09325296,50.040718323,483.103930387],[0.132670971,-0.022575789,0.326351779,-0.935619187],[-1,0,1,4],[134.887718951,9E+09,9E+09,9E+09,9E+09,9E+09]];
  CONST robtarget pAngerL_60:=[[396.062972248,27.911166703,492.703033028],[0.114272503,-0.022558134,0.275782172,-0.954136845],[-1,0,1,4],[129.639362388,9E+09,9E+09,9E+09,9E+09,9E+09]];
  CONST robtarget pContemptL_10:=[[-94.491553607,225.077568886,137.327093089],[0.306193092,0.231227469,-0.892125882,-0.238518467],[-1,0,1,5],[170.068678796,9E+09,9E+09,9E+09,9E+09,9E+09]];
  CONST robtarget pToDissL_10:=[[311.262788205,141.365155063,320.620976131],[0.30127594,0.413850338,-0.12183377,0.850363004],[-1,0,0,4],[109.137922493,9E+09,9E+09,9E+09,9E+09,9E+09]];
  CONST robtarget pToDissL_20:=[[313.163869898,99.550091581,313.678214603],[0.405584331,0.369718383,-0.180052484,0.816327612],[-1,0,0,4],[120.550323233,9E+09,9E+09,9E+09,9E+09,9E+09]];
  CONST robtarget pToDissL_30:=[[327.793203037,3.134311337,277.462215839],[0.525517576,0.35593926,-0.443885036,0.632538216],[-1,0,0,4],[161.707001678,9E+09,9E+09,9E+09,9E+09,9E+09]];
  CONST robtarget pToDissL_40:=[[274.023321791,-80.991562457,305.086937965],[0.647848865,0.227051384,-0.451204352,0.570222895],[-1,0,0,4],[171.12747593,9E+09,9E+09,9E+09,9E+09,9E+09]];
  CONST robtarget pToDissL_50:=[[233.086731165,-187.421735572,361.300083015],[0.647848463,0.227050931,-0.451204503,0.570223413],[-1,1,-1,4],[154.498524311,9E+09,9E+09,9E+09,9E+09,9E+09]];
  VAR syncident syncToDiss;
  CONST robtarget pSuprisedL_10:=[[108.153191894,471.411528047,647.230762026],[0.699371757,0.003098078,0.006552088,-0.714721357],[-1,0,0,4],[-132.382826108,9E+09,9E+09,9E+09,9E+09,9E+09]];
  CONST robtarget pHandsUpL_10:=[[108.153567372,471.411547841,988.720364525],[0.699371728,0.003098049,0.006552252,-0.714721384],[0,-1,0,4],[-132.382818416,9E+09,9E+09,9E+09,9E+09,9E+09]];
  CONST robtarget pNoClueL_20:=[[332.599072052,360.424339744,333.84998915],[0.323491568,-0.733582932,-0.040436016,-0.596300441],[-1,0,0,5],[100.391786771,9E+09,9E+09,9E+09,9E+09,9E+09]];
  CONST robtarget pNoClueL_10:=[[116.844170561,567.745373907,549.176802943],[0.612414859,-0.27944775,-0.40047322,-0.621673705],[-1,0,0,5],[170.97345488,9E+09,9E+09,9E+09,9E+09,9E+09]];
  CONST robtarget pGiveMeAHug10:=[[527.97,296.13,502.72],[0.151847,-0.178758,0.845099,-0.480413],[0,0,0,4],[-148.435,9E+09,9E+09,9E+09,9E+09,9E+09]];
  VAR syncident syncGiveMeAHug;
  CONST robtarget pGiveMeAHug20:=[[405.4,271.24,496.02],[0.213733,-0.0269022,-0.854052,0.473487],[0,0,0,4],[-149.626,9E+09,9E+09,9E+09,9E+09,9E+09]];
  VAR syncident syncGiveMeAHug1;
  VAR syncident syncGoAway;
  CONST robtarget pGoAway10:=[[201.45,40.13,222.49],[0.507555,0.594761,-0.385316,0.49008],[0,1,-1,4],[118.012,9E+09,9E+09,9E+09,9E+09,9E+09]];
  CONST robtarget pGoAway20:=[[518.18,74.7,248.67],[0.288596,0.590195,-0.341764,0.671997],[-1,1,-1,4],[116.115,9E+09,9E+09,9E+09,9E+09,9E+09]];
  VAR syncident syncGoAway1;
  VAR syncident syncGoAway2;
  CONST robtarget pPowerfull10:=[[118.3,247.25,704.02],[0.422171,0.460914,0.546915,-0.556969],[-1,0,0,4],[179.781,9E+09,9E+09,9E+09,9E+09,9E+09]];
  CONST robtarget pPowerfull20:=[[245.96,143,310.92],[0.0443739,-0.318911,0.39353,-0.861081],[0,0,0,4],[112.918,9E+09,9E+09,9E+09,9E+09,9E+09]];
  CONST robtarget pPowerfull30:=[[252,-77.89,315.69],[0.488544,0.342198,-0.661481,0.454609],[-1,1,-1,4],[123.612,9E+09,9E+09,9E+09,9E+09,9E+09]];
  CONST robtarget pPowerfull40:=[[322,-67.67,364.23],[0.442195,0.413994,-0.46771,0.643677],[-1,1,-1,4],[123.892,9E+09,9E+09,9E+09,9E+09,9E+09]];
  VAR syncident syncPowerfull;
  CONST robtarget pHappy10:=[[139.69,626.34,927.43],[0.90409,-0.412355,0.0928741,-0.0629285],[0,0,0,6],[-47.2014,9E+09,9E+09,9E+09,9E+09,9E+09]];
  VAR syncident syncHappy;
  CONST robtarget pHappy20:=[[263.63,23.73,371.01],[0.080959,0.0864927,-0.709647,0.694526],[0,0,0,4],[-174.693,9E+09,9E+09,9E+09,9E+09,9E+09]];
  VAR syncident syncHappy1;
  VAR syncident syncHappy2;
  CONST robtarget pHappy30:=[[298.49,-216.51,440.95],[0.379184,0.0939631,-0.443299,0.806769],[-1,0,0,4],[153.776,9E+09,9E+09,9E+09,9E+09,9E+09]];
  VAR syncident syncHappy3;
  CONST robtarget pExcited10:=[[283.05,206.57,132.91],[0.0344361,0.707983,-0.0555807,0.703197],[0,0,0,4],[118.262,9E+09,9E+09,9E+09,9E+09,9E+09]];
  VAR syncident syncExcited;
  CONST robtarget pExcited20:=[[282.98,206.6,184.63],[0.0343905,0.708084,-0.0557234,0.703086],[0,0,0,4],[118.259,9E+09,9E+09,9E+09,9E+09,9E+09]];
  VAR syncident syncExcited1;
  CONST robtarget pExcited30:=[[327.61,77.77,391.45],[0.471456,0.494579,0.520471,-0.512085],[-1,1,0,4],[115.029,9E+09,9E+09,9E+09,9E+09,9E+09]];
  VAR syncident syncExcited2;
  CONST robtarget pExcited40:=[[327.81,34.51,391.34],[0.471431,0.494263,0.520659,-0.512222],[-1,1,0,4],[115.022,9E+09,9E+09,9E+09,9E+09,9E+09]];
  VAR syncident syncExcited3;
  CONST robtarget pScared10:=[[253.81,59.02,495.38],[0.715734,-0.00275996,-0.0560464,0.696115],[-1,0,-1,4],[114.586,9E+09,9E+09,9E+09,9E+09,9E+09]];
  VAR syncident syncScared;
  CONST robtarget pScared20:=[[253.81,59.02,394.12],[0.715731,-0.00275244,-0.0560455,0.696118],[-1,0,-1,4],[114.588,9E+09,9E+09,9E+09,9E+09,9E+09]];
  VAR syncident syncScared1;
  PROC Home()
    MoveJ pHomeL_10,v1000,fine,Servo\WObj:=wobj0;
  ENDPROC
  PROC Contempt()
    WaitSyncTask syncCommandStart,task_list\TimeOut:=5;
    MoveJ pContemptL_10,v1000,fine,Servo\WObj:=wobj0;
    WaitTime 2;
    Home;
  ENDPROC
  PROC ToDiss()
    WaitSyncTask syncCommandStart,task_list\TimeOut:=5;
    MoveJ pToDissL_10,v1000,z10,Servo\WObj:=wobj0;
    MoveJ pToDissL_20,v1000,z10,Servo\WObj:=wobj0;
    MoveJ pToDissL_30,v1000,z10,Servo\WObj:=wobj0;
    MoveJ pToDissL_40,v1000,z10,Servo\WObj:=wobj0;
    MoveJ pToDissL_50,v1000,fine,Servo\WObj:=wobj0;
    WaitSyncTask syncToDiss,task_list;
    WaitTime 1;
    Home;
  ENDPROC
  PROC Suprised()
    WaitSyncTask syncCommandStart,task_list\TimeOut:=5;
    MoveJ pSuprisedL_10,v5000,fine,Servo\WObj:=wobj0;
    WaitTime 2;
    Home;
  ENDPROC
  PROC HandsUp()
    WaitSyncTask syncCommandStart,task_list\TimeOut:=5;
    MoveJ pHandsUpL_10,v1000,fine,Servo\WObj:=wobj0;
    WaitTime 2;
    Home;
  ENDPROC
  PROC NoClue()
    WaitSyncTask syncCommandStart,task_list\TimeOut:=5;
    MoveJ pNoClueL_20,v1000,z10,Servo\WObj:=wobj0;
    MoveJ pNoClueL_10,v1000,fine,Servo\WObj:=wobj0;
    WaitTime 2;
    MoveJ pNoClueL_20,v1000,z10,Servo\WObj:=wobj0;
    Home;
  ENDPROC
  PROC GiveMeAHug()
    MoveJ pGiveMeAHug10,v1000,fine,Servo;
    WaitSyncTask syncGiveMeAHug,task_list;
    WaitTime 2;
    MoveJ pGiveMeAHug20,v1000,fine,Servo;
    MoveJ pGiveMeAHug10,v1000,fine,Servo;
    MoveJ pGiveMeAHug20,v1000,fine,Servo;
    MoveJ pGiveMeAHug10,v1000,fine,Servo;
    MoveJ pGiveMeAHug20,v1000,fine,Servo;
    MoveJ pGiveMeAHug10,v1000,fine,Servo;
    MoveJ pGiveMeAHug20,v1000,fine,Servo;
    WaitSyncTask syncGiveMeAHug1,task_list;
    WaitTime 2;
    Home;
  ENDPROC
  PROC GoAway()
    WaitSyncTask syncCommandStart,task_list\TimeOut:=5;
    SyncMoveOn syncGoAway,task_list;
    MoveJ pGoAway10\ID:=10,v1000,fine,Servo;
    MoveJ pGoAway20\ID:=20,v1000,fine,Servo;
    MoveJ pGoAway10\ID:=30,v1000,fine,Servo;
    MoveJ pGoAway20\ID:=40,v1000,fine,Servo;
    MoveJ pGoAway10\ID:=50,v1000,fine,Servo;
    SyncMoveOff syncGoAway1;
    WaitSyncTask syncGoAway2,task_list;
    Home;
  ENDPROC
  PROC Powerful()
    WaitSyncTask syncCommandStart,task_list\TimeOut:=5;
    MoveJ pPowerfull10,v1000,fine,Servo;
    WaitTime 2;
    MoveJ pPowerfull20,v1000,fine,Servo;
    WaitTime 2;
    MoveJ pPowerfull30,v1000,fine,Servo;
    MoveJ pPowerfull40,v1000,fine,Servo;
    MoveJ pPowerfull30,v1000,fine,Servo;
    MoveJ pPowerfull40,v1000,fine,Servo;
    MoveJ pPowerfull30,v1000,fine,Servo;
    MoveJ pPowerfull20,v1000,fine,Servo;
    WaitTime 2;
    WaitSyncTask syncPowerfull,task_list;
    Home;
  ENDPROC
  PROC Happy()
    WaitSyncTask syncCommandStart,task_list\TimeOut:=5;
    MoveJ pHappy10,v1000,fine,Servo;
    WaitTime 1;
    WaitSyncTask syncHappy,task_list;
    MoveJ pHappy20,v1000,fine,Servo;
    SyncMoveOn syncHappy1,task_list;
    MoveC Offs(pHappy20,nCircleDiameter/2, 0, nCircleDiameter/2),Offs(pHappy20,nCircleDiameter, 0, 0)\ID:=10,v1000,z5,Servo;
    MoveC Offs(pHappy20,nCircleDiameter/2, 0, -nCircleDiameter/2),pHappy20\ID:=20,v1000,z5,Servo;
    MoveC Offs(pHappy20,nCircleDiameter/2, 0, nCircleDiameter/2),Offs(pHappy20,nCircleDiameter, 0, 0)\ID:=30,v1000,z5,Servo;
    MoveC Offs(pHappy20,nCircleDiameter/2, 0, -nCircleDiameter/2),pHappy20\ID:=40,v1000,z5,Servo;
    SyncMoveOff syncHappy2;
    MoveJ pHappy30,v1000,fine,Servo;
    WaitTime 2;
    WaitSyncTask syncHappy3,task_list;
    Home;
  ENDPROC
  PROC Excited()
    WaitSyncTask syncCommandStart,task_list\TimeOut:=5;
    MoveJ pExcited10,v1000,fine,Servo;
    SyncMoveOn syncExcited,task_list;
    MoveJ pExcited20\ID:=10,v1000,z5,Servo;
    MoveJ pExcited10\ID:=20,v1000,z5,Servo;
    MoveJ pExcited20\ID:=30,v1000,z5,Servo;
    MoveJ pExcited10\ID:=40,v1000,z5,Servo;
    MoveJ pExcited20\ID:=50,v1000,z5,Servo;
    MoveJ pExcited10\ID:=60,v1000,fine,Servo;
    SyncMoveOff syncExcited1;
    WaitTime 1;
    MoveJ pExcited30,v1000,fine,Servo;
    WaitTime 0.5;
    SyncMoveOn syncExcited2,task_list;
    MoveJ pExcited40\ID:=10,v1000,z5,Servo;
    MoveJ pExcited30\ID:=20,v1000,z5,Servo;
    MoveJ pExcited40\ID:=30,v1000,z5,Servo;
    MoveJ pExcited30\ID:=40,v1000,z5,Servo;
    MoveJ pExcited40\ID:=50,v1000,z5,Servo;
    MoveJ pExcited30\ID:=60,v1000,fine,Servo;
    SyncMoveOff syncExcited3;
    WaitTime 2;
    Home;
  ENDPROC
  PROC Scared()
    WaitSyncTask syncCommandStart,task_list\TimeOut:=5;
    MoveJ pScared10,v1000,fine,Servo;
    WaitTime 2;
    SyncMoveOn syncScared,task_list;
    MoveJ pScared20\ID:=10,v100,fine,Servo;
    MoveJ pScared10\ID:=20,v1000,fine,Servo;
    SyncMoveOff syncScared1;
    WaitTime 2;
    Home;
  ENDPROC
ENDMODULE

! task T_ROB_L
MODULE Gripper_L
  PERS tooldata Servo:=[TRUE,[[0,0,114.2],[1,0,0,0]],[0.24,[8.2,12.5,48.1],[1,0,0,0],0.00022,0.00024,0.00009]];
ENDMODULE

! task T_ROB_L
MODULE MainModule
  PERS tasks task_list{2};
ENDMODULE

